// TIA Portal V17 export
// export: Created 2025-01-08T13:55:36.3322541Z, ExportSetting WithDefaults, DisplayName Totally Integrated Automation Portal, DisplayVersion V17, DisplayName TIA Portal Openness, DisplayVersion V17, DisplayName TIA Portal Version Control Interface, DisplayVersion V17, DisplayName SINAMICS Startdrive Advanced, DisplayVersion V17 Update2, DisplayName SINAMICS Startdrive G130, G150, S120, S150, SINAMICS MV, S210, DisplayVersion V17 Update2, DisplayName SINAMICS Startdrive G110M, G120, G120C, G120D, G120P, G115D, DisplayVersion V17 Update2, DisplayName STEP 7 Professional, DisplayVersion V17, DisplayName STEP 7 Safety, DisplayVersion V17, DisplayName WinCC Advanced, DisplayVersion V17
TYPE "DataToHSM"
// stored: IsFailsafeCompliant false
   STRUCT
      Cmd : Struct   // Command Send
         xStop : Bool;   // Offline
         xRun : Bool;   // Online
         xService : Bool;
         xTeach : Bool;
         xFeed : Bool;
         xSaveConfiguration : Bool;   // Reserved but not used for the time being
         xLoadConfiguration : Bool;   // Reserved but not used for the time being
         xRecieveContent : Bool;   // Reserved but not used for the time being
         xCparameterSend : Bool;   // Starts sending all K parameters selected via Kparameter mask to the labeling system / Starts sending all C parameters selected via C parameter mask to the labeling system
         xCparameterReceive : Bool;   // Requests the labeling system to send all parameters
         xMparameterSend : Bool;   // Starts sending all the M parameters selected via the Mparameter mask to the labeling system
         xMparameterReceive : Bool;   // Requests all labeling parameters to be sent from the labeling system
         xReserve : Bool;
         xReceiveTime : Bool;
         xGetMACandFWversion : Bool;
         xActivateContinuousStatus : Bool;   // 1: Activates the continuous transfer of the control register (initially not used)
         xWatchDog : Bool;   // Sign of Life Bit
         xAcknowledgeFaultFromExternal : Bool;   // PLC can directly acknowledge a malfunction of the labeling system
         xBlockProductPhotocell : Bool;   // 1: Product sensor is not active, i.e. no labeling pulse is triggered
         "xSplice-Start" : Bool;
         xReserved_19 : Bool;
         xReserved_18 : Bool;
         xReserved_17 : Bool;
         xReserved_16 : Bool;
         xReserved_15 : Bool;
         xReserved_14 : Bool;
         xReserved_13 : Bool;
         xReserved_12 : Bool;
         xReserved_11 : Bool;
         xReserved_10 : Bool;
         xReserved_09 : Bool;
         xReserved_08 : Bool;
         ParaMask : "HSMConfigAndMachineParameterMask";
         iUpdateRate : Int;   // Rate in ms at which the control register is updated
         iReserved_03 : Int;
         iReserved_02 : Int;
         iReserved_01 : Int;
      END_STRUCT;
      Cfg : Struct   // Configuration Parameters Send
         iDesiredInternalSpeed : Int;   // in 1/10 m / min (desired speed value)
         iDispenseDelay : Int;   // in 1/10 mm
         iLabelPosition : Int;   // in 1/10 mm
         iLabelLength : Int;   // in mm
         iLabelGap : Int;   // in 1/10 mm
         iLabelBurst : Int;   // 1 = off, 2 = twice ... (several labels with one trigger pulse)
         iLabelDistance : Int;   // in 1/10 mm (distance between the labels if several per trigger)
         iMaxNumberOfLabelSkips : Int;   // 0 - n
         iTriggerBlanking : Int;   // in mm
         iAccelerationRamp : Int;   // in 1/10 mm
         iSpeedInternalOrEncoder : Int;   // 0 = internal, 1 = encoder
         iStopRamp : Int;   // in% (ratio to acceleration ramp)
         iSyncOutputDelay : Int;   // in 1/10 mm
         iSyncOutputLenght : Int;   // in 1/10 mm
         iSyncOutput2Delay : Int;   // in 1/10 mm
         iSyncOutput2Lenght : Int;   // in 1/10 mm
         iSyncOutput3Delay : Int;   // in 1/10 mm
         iSyncOutput3Lenght : Int;   // in 1/10 mm
         iPreFeedLenght : Int;   // in 1/10 mm
         iConveyorSpeed_1 : Int;
         iConveyorSpeed_2 : Int;
         iReserved_11 : Int;
         iReserved_10 : Int;
         iReserved_09 : Int;
         iReserved_08 : Int;
         iReserved_07 : Int;
         iReserved_06 : Int;
         iReserved_05 : Int;
         iReserved_04 : Int;
         iReserved_03 : Int;
         iReserved_02 : Int;
         iReserved_01 : Int;
      END_STRUCT;
      MPar : Struct   // Machine Parameters Send
         iSpeedInternalOrEncoder : Int;   // 0 = Fixed internally, 1 = Encoder fixed, 2 = Value from configuration
         iDistancePerEncoderRevolution : Int;   // in 1/10 mm
         iPulsesPerEncoderRevolution : Int;   // in Pulse
         iMaxSpeed : Int;   // in 1/10 m/min
         iInstallationsMode : Int;   // 0 = normal, 1 = feed also via start button, 2 = feed with fixed length via start button, 3 = feed always with fixed length
         iBackingPaperLengthPerMotorRevolution : Int;   // in 1/100 mm
         iDistanceToDispensingEdgeToGapSensor : Int;   // in 1/10 mm (required for changeable dispense tongues and changed depending on the product)
         iProductsensorPolarity : Int;   // 0 = NPN, 1 = NPN inverted, 2 = PNP inverted, 3 = PNP
         iSkipMode : Int;   // 0 = value from configuration, 1 = value from machine parameters, 2 = end detect
         iMaxNumberOfLabelSkips : Int;   // 0 - n
         iAccelerationRampMode : Int;   // 0 = value from configuration, 1 = value from machine parameters
         iAccelerationRamp : Int;   // in 1/10 mm
         iGapSensor : Int;   // 0 = leading edge, 1 = trailing edge label
         iMaxCalibrationDistance : Int;   // in 1/10mm
         iDecelerationRampMode : Int;   // 0 = value from configuration, 1 = value from machine parameters
         iDecelerationRamp : Int;   // in% (ratio to acceleration ramp)
         iExternalStart : Int;   // 0 = off 1 = edge controlled 2 = pulse controlled
         iLowLabelInput : Int;   // 0 = off 1 = on
         iRibbonInput : Int;   // 0 = off 1 = on
         iSyncParameter : Int;   // 0 = value from configuration, 1 = value from machine parameters
         iSyncOutputDelay : Int;   // in 1/10mm
         iSyncOutputLenght : Int;   // in 1/10mm
         iZeroDownTimeMode : Int;   // 0 = Off 1 = Master 2 = Slave
         iZeroDownTimeSensorDistance : Int;   // in mm
         iRestLenghtOnLowLabel : Int;   // in m
         iLowLabelSensorPolarity : Int;   // 2 = PNP inverted 3 = PNP
         iWebBreakSensorPolarity : Int;   // 2 = PNP inverted 3 = PNP
         iWarningOutputPolarity : Int;   // 2 = PNP inverted 3 = PNP
         iSync2Parameter : Int;   // 0 = value from configuration, 1 = value from machine parameters
         iSync2OutputDelay : Int;   // in 1/10mm
         iSync2OutputLenght : Int;   // in 1/10mm
         iSync3Parameter : Int;   // 0 = value from configuration, 1 = value from machine parameters
         iSync3OutputDelay : Int;   // in 1/10mm
         iSync3OutputLenght : Int;   // in 1/10mm
         iTeachTolerance : Int;   // in 1/100mm
         iSynch1Mode : Int;   // 0 = production sensor 1 = trigger sensor 2 = reserve 3 = end of dispense
         iSynch2Mode : Int;   // 0 = production sensor 1 = trigger sensor 2 = reserve 3 = end of dispense
         iSynch3Mode : Int;   // 0 = production sensor 1 = trigger sensor 2 = reserve 3 = end of dispense
         iOverCurrentCorrection : Int;   // in %
         iServiceFeedRate : Int := 10;   // in 1/10 m/min
         iPreFeedMode : Int;   // 0 = value from configuration, 1 = value from machine parameters
         iPreFeed : Int;   // in 1/10 mm
         iLabelSensorWindowPreFeedLenght : Int;   // in 1/10 mm
         iLabelSensorCount : Int;
         "iSPS-Mode" : Int;   // 0= Off 1= S7-Kommunikation / 0= Off 1= S7-communication, 2 = S7-communication double size
         iZdtWin : Int;   // Zero Down Time Window mm
         iDistRes : Int;   // Resolution label spacing
         "iSPS-DB-No-Ctrl" : Int;   // Data block for PLC communication
         "iSPS-DB-No-Stat" : Int;   // Data block for PLC communication
         iSignalFormat : Int;   // Is relevant for the WEBER-TOOL
         iLowLabDiam : Int;   // Roll diameter for LowLab in 1/10 mm
         iCoreDiameter : Int;   // Core diameter in 1/10 mm
         iWebBreakRest : Int;   // Rest after WebBreak in mm
         iLeverSetup : Int;   // To the TEACH of the dancer position
         iLeverMinPos : Int;   // Analog value angle sensor unwinder dancer Min.Pos.
         iLeverMaxPos : Int;   // Analog value angle sensor unwinder dancer Max.Pos.
         "iUW-BufLength" : Int;   // Label path in mm between dancers min / max
         iTwinLabelMd : Int;   // Double Label mode
         iLabQueuwTolerance : Int := 10;   // Setting the tolerance "Number of labels between peel bar and label sensor".
         iResetEvents : Int;   // Reset the operating data EV#007 „Number of all spent labels“ or EV#008 „Display of label roll dispensed“. 0 = off, 1 = reset EV#007 Label feeds, 2 = reset EV#008 Label meters.
         iMaintananceDistancekm : Int;   // Setting the maintenance interval depending on the the label roll length. [km]
         iMaintananceDays : Int;   // Setting the maintenance interval depending on the operation time. [days]
         iProductSensorMode : Int;   // Defines the linkage of the product sensors 1 and 2 with respect to the trigger signal. 0 = Off, 1 = AND Operation (both sensors must recieve a signal), 2 = OR operation (only one sensor have to recieve a signal)
         iRewinderDiameterWarning : Int := 2600;   // Defines the diameter of the carrier web, after which a pre-warning for the rewinder is avti-vated. The following message appears "Rewinder almost full".
         iRewinderDiameterFull : Int := 2650;   // Defines the diameter of the carrier web, after which the labeler stops. The following mes-sage appears "Rewinder full".
         iMotorLoadLimit : Int := 90;   // Defines the value for the motor current, after which the following message appears "Load approaching the upper limit".
         iContourRamp : Int;   // Parameter for activating contour mode. When the parameter is activated, the two parameters "Start contour" and "Stop contour" are displayed in the configuration menu. At the same time, the "Ramp" parameter is ignored.
         iEncoderOutPulsPermm : Int;   // Determines the number of encoder pulses per millimeter of label path and synchronizes an optional printer at the AUX socket.
         iPLCRackAndSlot : Int := 10;   // This Parameter is used to set the communication with different PLC versions.
         iSliceDistance : Int := 2000;   // This parameter is used to set the distance (duration) in splice mode. The label web is ad-vanced with the reduced speed specified in parameter 071. 0 - 9999. Adjusting the value in [mm]
         iSpliceSpeedReduction : Int := 33;   // This parameter is only used if parameter 070 is active. It is used to reduce reduce the speed in the slice mode and is calculated on the basis of the current speed. 10 - 100. Adjusting the value in [%]
         iDownstream : Int := 20;   // This parameter is only used for alternating operation and defines the transfer reserve that is still to be dispensed in alternating operation. Must be less than or equal to Par.25 RestLowLabel. 0.0 – 90.0. Adjusting the value in [m]
         iSpeedFactor : Int := 1000;   // Offset setting for operation with rotary encoder. The feed rate of the dispenser is factor Par.73 x encoder speed. 20.0 - 500.0. Adjusting the value in [%].
         iAcceleration : Int;   // Setting of the start ramp setting in m/s2. If the value is 0, the ramp length is used to calcu-late the acceleration. The stop ramp is set exactly as before via the ratio to the start ramp. 0.0 - 90.0. In [m/s2]
         iSpeedOffset : Int;   // Setting of a speed offset in 1/10 m/min. Only applies to the internal speed. Parameter 073 can be used in encoder mode. -20.0 - 20.0. in [%]
         iMaterialTransportErrorMode : Int;   // Determines whether the material transport error "Materialtransportoffen" is to be output. The signal for the error must be applied to X22.4. 0 = Off. 1 = Error at 24V. 2 = Error at 0V.
         iEncoderFactor : Int := 1000;   // Offset setting of the encoder speed for the internal calculation of Alpha HSM, e.g. for win-ding tape operation and ZDT application. Alpha HSM must calculate with baseband speed for the function of the ZDT, but dispenses with encoder speed from the winding belt. 20.0 - 500.0. In [%]
         Reserve_1 : Int;
         Reserve_2 : Int;
         Reserve_3 : Int;
         Reserve_4 : Int;
         Reserve_5 : Int;
         Reserve_6 : Int;
         Reserve_7 : Int;
         Reserve_8 : Int;
         Reserve_9 : Int;
         Reserve_10 : Int;
         Reserve_11 : Int;
         Reserve_12 : Int;
         Reserve_13 : Int;
         Reserve_14 : Int;
         Reserve_15 : Int;
         Reserve_16 : Int;
         Reserve_17 : Int;
         Reserve_18 : Int;
         Reserve_19 : Int;
         Reserve_20 : Int;
         Reserve_21 : Int;
         Reserve_22 : Int;
         Reserve_23 : Int;
         Reserve_24 : Int;
         Reserve_25 : Int;
         Reserve_26 : Int;
         Reserve_27 : Int;
         Reserve_28 : Int;
         Reserve_29 : Int;
         Reserve_30 : Int;
         Reserve_31 : Int;
         Reserve_32 : Int;
         Reserve_33 : Int;
         Reserve_34 : Int;
         Reserve_35 : Int;
         Reserve_36 : Int;
         Reserve_37 : Int;
         Reserve_38 : Int;
         Reserve_39 : Int;
         Reserve_40 : Int;
         Reserve_41 : Int;
         Reserve_42 : Int;
         Reserve_43 : Int;
         Reserve_44 : Int;
         Reserve_45 : Int;
         Reserve_46 : Int;
         Reserve_47 : Int;
         Reserve_48 : Int;
         Reserve_49 : Int;
         Reserve_50 : Int;
         Reserve_51 : Int;
      END_STRUCT;
   END_STRUCT;
END_TYPE
